FUNCTION_BLOCK MUX_SINT (* See MUX_ANY *)
  (* Standard: 61131-3 *)
  (* Version 0.0, 2004-12-15, JHC, Rockwell Automation, Converted from SRC format. *)
  (* Compiler header: package fb.rt.plc.select; *)
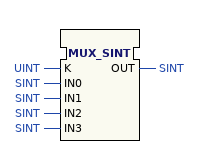
  VAR_INPUT
    K : UINT;
    IN0 : SINT;
    IN1 : SINT;
    IN2 : SINT;
    IN3 : SINT;
  END_VAR
  VAR_OUTPUT
    OUT : SINT;
  END_VAR
END_FUNCTION_BLOCK
